PROGRAM P_Control_Mode
VAR
END_VAR


// ***********************************************************************************
//
// USI Mendrisio, Largo Bernasconi 2, CH-6850 Mendrisio
// ETH Zurich, Building HIF E26, Laura-Hezner-Weg 7, CH-8093 Zürich
//
// ***********************************************************************************
//
// PROJECT     :  Clay Printing Controller
// FUNCTION    :  Control mode selection
// AUTHOR      :  WeiTing Chen
// EMAIL       :  chen@mesh.ch
// Copyright   :  USI FMAA Mendrisio(CH) 2025
//
// ***********************************************************************************


GVL.b_mode_manual := GVL_IO.ib_CC1_Button_Mode_Manual;
GVL.b_mode_laptop := GVL_IO.ib_CC1_Button_Mode_Laptop;
GVL.b_mode_robot := False;

IF GVL.b_mode_manual THEN
	GVL.s_current_mode := 'Controller';
ELSIF GVL.b_mode_laptop  THEN
	GVL.s_current_mode := 'Laptop';
// if all not run robot mode
ELSIF NOT GVL.b_mode_manual AND NOT GVL.b_mode_laptop THEN
	GVL.s_current_mode := 'Robot';
	GVL.b_mode_robot := TRUE;
ELSE
	GVL.s_current_mode := 'None';

END_IF

END_PROGRAM

(* stored: Version 1.1.0.1, ProductVersion 3.1.4024.15
   POU P_Control_Mode: Id {257c4f21-4afb-49d3-84fe-3325b52e1ec9}, SpecialFunc None *)
